FUNCTION_BLOCK TestSocketAndPlug (* Template for a simple Basic Function Block Type *)
  (* Standard: 61499-2; Description: Copyright (c) 2019 Jan Holzweber This program and the accompanying materials are made available under the terms of the Eclipse Public License 2.0 which is available at https://www.eclipse.org/legal/epl-2.0/ SPDX-License-Identifier: EPL-2.0 *)
  (* Version 1.0, 2019-07-25, Jan Holzweber *)
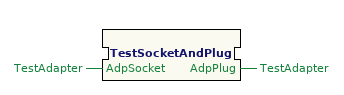
  SOCKETS
    AdpSocket : TestAdapter;
  END_SOCKETS
  PLUGS
    AdpPlug : TestAdapter;
  END_PLUGS
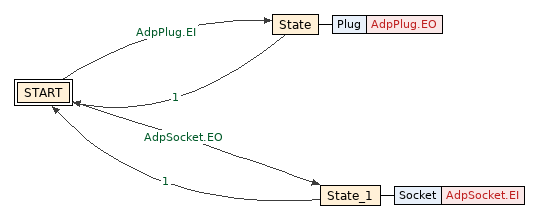
  EC_STATES
    START; (* Initial State *)
    State : Plug -> AdpPlug.EO;
    State_1 : Socket -> AdpSocket.EI;
  END_STATES
  EC_TRANSITIONS
    START TO State := AdpPlug.EI;
    State TO START := 1;
    START TO State_1 := AdpSocket.EO;
    State_1 TO START := 1;
  END_TRANSITIONS
  ALGORITHM Plug IN ST: (* new algorithm *)
AdpPlug.D0 := AdpPlug.DI;
  END_ALGORITHM
  ALGORITHM Socket IN ST: (* new algorithm *)
AdpSocket.DI := AdpSocket.D0;
  END_ALGORITHM
END_FUNCTION_BLOCK
